Staubli VAL3: remSetMaxA.pgx

program remSetMaxA(string& sArgs[] (dimensions=1), string& sReturn[] (dimensions=1))
  local num bOk
  local num nVal
begin
  // Set the maximum allowed Acceleration in %
  //
  logMsg("call remSetMaxA")
  call remSetnGlobal(sArgs,nMaxAccel,0,100,"SETMAXA",sReturn)
end
